FUNCTION_BLOCK DoubleCylinderBaseTestContext EXTENDS TcoCore._internals_TcoContext
VAR
    _sut : DoubleCylinderBaseImplemented(THIS^);
    _sutInvalid : DoubleCylinderBaseImplemented(THIS^);
    _atHomeSignal : BOOL;
    _atWorkSignal : BOOL;
    _toHomeSignal : BOOL;
    _toWorkSignal : BOOL;
END_VAR
VAR
    _get_AtHome : BOOL;
    _get_AtWork : BOOL;
END_VAR

METHOD PROTECTED Main
_sut(inoAtHomePos1 := _atHomeSignal,
    inoAtHomePos2 := _atHomeSignal,
    inoAtWorkPos1 := _atWorkSignal,
    inoAtWorkPos2 := _atWorkSignal,
    inoToHomePos := _toHomeSignal,
    inoToWorkPos := _toWorkSignal);

CASE _testId OF
    eCyclinderBaseTests.Invalid:
        _sutInvalid.AtHome;
        _sutInvalid.AtWork;
        _sutInvalid.Restore();
        _sutInvalid.Stop();
    eCyclinderBaseTests.GetAtHome:
        _get_AtHome := _sut.AtHome;
    eCyclinderBaseTests.GetAtWork:
        _get_AtWork := _sut.AtWork;
END_CASE
END_METHOD

END_FUNCTION_BLOCK

(* stored: Version 1.1.0.1, ProductVersion 3.1.4024.10
   POU DoubleCylinderBaseTestContext: Id {d872de45-e829-05c4-2cef-dfad02f8f7a2}, SpecialFunc None
   Method Main: Id {6480da05-d898-0bdf-317f-5e0e346c2889} *)
